FUNCTION_BLOCK FB_CleaningProcessStateBase
VAR_INPUT
  I_ParentCallback : I_CleaningStateCallback;
  I_MachineStatus  : I_MachineStateBase;
END_VAR

VAR_OUTPUT
END_VAR

VAR
  sL_StateName	 : STRING;
	
  //Device operation
  iL_CurrentStep : INT;
  iL_State       : INT := 1;
  bL_DevOpActive : BOOL;
  bL_AbortPend   : BOOL;
END_VAR

VAR_STAT
  bL_InitDone    : BOOL := FALSE;
END_VAR	

VAR CONSTANT
  //Device operation
  cL_SEND    : INT := 1;
  cL_WAIT    : INT := 2;	
  cL_NEXT    : INT := 3;	
  cL_DONE    : INT := 4;
  cL_ERROR   : INT := 5;

  cL_MaxStep : INT := 15; //Make dynamic one day	
END_VAR

//No code here, use mStateAction

METHOD mAbort : BOOL
VAR_INPUT
END_VAR
IF NOT bL_AbortPend THEN
  I_ParentCallback.mDeviceAbort();
  bL_AbortPend:=TRUE;
  
  IF NOT bL_DevOpActive THEN
    bL_DevOpActive := TRUE; //Set to relaunch process
    iL_CurrentStep := 0;
	END_IF
END_IF
END_METHOD

METHOD mAckError : BOOL
VAR_INPUT
END_VAR
END_METHOD

METHOD mCleaningOp : BOOL
VAR_INPUT
	sI_Operation : EN_CLEANING_OP;
END_VAR
//Service not implemented
mCleaningOp:=FALSE;
END_METHOD

METHOD mDevOp
VAR_INPUT
END_VAR

VAR
  sL_Status : ST_CLEANING_DEV_STATUS;
END_VAR
sL_Status := I_ParentCallback.pDeviceStatus;
I_ParentCallback.mDeviceOperation(iL_CurrentStep);

CASE iL_State OF
  // Send command to devices
  cL_SEND:
    iL_State := cL_WAIT;  
    
  // Wait until operation completed  
  cL_WAIT:
    IF sL_Status.bError THEN
      iL_State := cL_ERROR;
    ELSIF NOT sL_Status.bBusy THEN
      iL_State := cL_NEXT;
    END_IF
    
  // Next state 
  cL_NEXT:
    IF iL_CurrentStep < cL_MaxStep AND NOT sL_Status.bReady THEN
      iL_CurrentStep := iL_CurrentStep + 1;  

      iL_State := cL_SEND;
    ELSE
      iL_State := cL_DONE;
    END_IF
    
  // Done
  cL_DONE:
    bL_DevOpActive := FALSE; //Clear cleaning flag
    iL_State       := cL_SEND; //Init for next operation
    iL_CurrentStep := 0;
    I_ParentCallback.mSetMode(EN_CLEANING_OP.eNOP);
    mDevOpDone();
  
  // Error
  cL_ERROR:
    bL_DevOpActive := FALSE; //Clear cleaning flag
    iL_State       := cL_SEND; //Init for next operation
    iL_CurrentStep := 0;
END_CASE
END_METHOD

METHOD mDevOpDone : BOOL
VAR_INPUT
END_VAR
//Optional action when device operation completed

//Operation (incl. Abort) terminated
bL_AbortPend:=FALSE;
END_METHOD

METHOD mEntryAction
VAR_INPUT
END_VAR
END_METHOD

METHOD mExitAction
VAR_INPUT
END_VAR
END_METHOD

METHOD mInit : BOOL
VAR_INPUT
  I_parentMachineState : I_MachineStateBase;
  I_Callback           : I_CleaningStateCallback;
END_VAR
I_MachineStatus  := I_parentMachineState;
I_ParentCallback := I_Callback;
END_METHOD

METHOD mProduction : BOOL
VAR_INPUT
END_VAR
//Request production mode - implement in SubClass
mProduction := FALSE;
END_METHOD

METHOD mService : BOOL
VAR_INPUT
END_VAR
//Request service mode - implement in SubClass
mService := FALSE;
END_METHOD

METHOD mStateAction
VAR_INPUT
END_VAR

VAR
	sL_DeviceStatus: ST_CLEANING_DEV_STATUS;
END_VAR
sL_DeviceStatus := I_ParentCallback.pDeviceStatus;

//If a device has an error go to error state
IF sL_DeviceStatus.bError THEN
	I_ParentCallback.mChangeState(EN_Cleaning_State.Error);
END_IF
END_METHOD

PROPERTY pInitDone : BOOL
GET
pInitDone := bL_InitDone;
END_GET
SET
bL_InitDone := pInitDone;
END_SET
END_PROPERTY

PROPERTY pName : STRING
GET
pName := sL_StateName;
END_GET
SET
sL_StateName := pName;
END_SET
END_PROPERTY

END_FUNCTION_BLOCK

(* stored: Version 1.1.0.1, ProductVersion 3.1.4024.11
   POU FB_CleaningProcessStateBase: Id {1fb880ed-fc4b-4d4a-9b77-4e59ea92aa38}, SpecialFunc None
   Method mAbort: Id {9f866fbb-56cd-423a-b16e-c4d36a2d605e}
   Method mAckError: Id {ea120e02-a1f3-4acb-85c1-240606f9feb6}
   Method mCleaningOp: Id {162a8e04-79dc-42e2-9dd4-60348bfcb196}
   Method mDevOp: Id {c833d6e1-8c3d-4004-b63e-6c9f6b825475}
   Method mDevOpDone: Id {f0fd9669-d5d5-409f-bfec-43a15199ad59}
   Method mEntryAction: Id {21d00247-c914-4e71-914f-52455a25ef34}
   Method mExitAction: Id {5d83e7e7-be2f-435f-abe0-05fbca3be7d2}
   Method mInit: Id {837d1fff-8b3b-4ef1-933c-4d65379c6f1f}
   Method mProduction: Id {0cef4a27-1757-4a47-80ff-460f155c9faa}
   Method mService: Id {d60fbf11-a87b-4469-9b01-8e2871003aa3}
   Method mStateAction: Id {5a6548cd-2198-4689-be2a-fb5211cee55b}
   Property pInitDone: Id {5f863ae9-b141-45ca-b4b3-809572b1454a}
   Get Get: Id {5089d33b-e2fe-4875-b68e-88d13700f128}
   Set Set: Id {2db54f43-1a25-4343-8aab-a5d475c3efe5}
   Property pName: Id {1760e0d2-5f53-4226-89bc-29af38ecde9f}
   Get Get: Id {d3bc9210-7205-4570-9297-6047746ffa83}
   Set Set: Id {ee01f5fa-ae1e-45d6-999f-d63c2db63bc4} *)
